// TIA Portal V18 export
DATA_BLOCK "SS1_A8_16DI_16DO_DI_Vars"   // DB11081
{ S7_Optimized_Access := 'FALSE' }
VERSION : 0.1
// stored: AutoNumber false, DBAccessibleFromOPCUA true, IsOnlyStoredInLoadMemory false, IsWriteProtectedInAS false
   VAR
      DI1 : "UDT_DIadv";
      DI2 : "UDT_DIadv";
      DI3 : "UDT_DIadv";
      DI4 : "UDT_DIadv";
      DI5 : "UDT_DIadv";
      DI6 : "UDT_DIadv";
      DI7 : "UDT_DIadv";
      DI8 : "UDT_DIadv";
      DI9 { S7_SetPoint := 'True'} : "UDT_DIadv";
      DI10 { S7_SetPoint := 'True'} : "UDT_DIadv";
      DI11 { S7_SetPoint := 'True'} : "UDT_DIadv";
      DI12 { S7_SetPoint := 'True'} : "UDT_DIadv";
      DI13 { S7_SetPoint := 'True'} : "UDT_DIadv";
      DI14 { S7_SetPoint := 'True'} : "UDT_DIadv";
      DI15 { S7_SetPoint := 'True'} : "UDT_DIadv";
      DI16 { S7_SetPoint := 'True'} : "UDT_DIadv";
   END_VAR
BEGIN
   DI1.cFuncSystemID := 1;
   DI1.cFuncVar := 11;
   DI2.cFuncSystemID := 1;
   DI3.cFuncSystemID := 1;
   DI4.cFuncSystemID := 1;
   DI4.cFuncVar := 6;
   DI5.cFuncSystemID := 1;
   DI5.cFuncVar := 4;
   DI6.cFuncSystemID := 1;
   DI6.cFuncVar := 21;
   DI7.cFuncSystemID := 1;
   DI8.cFuncSystemID := 1;
   DI9.cFuncSystemID := 1;
   DI10.cFuncSystemID := 3;
   DI10.cFuncVar := 13;
   DI11.cFuncSystemID := 3;
   DI12.cFuncSystemID := 3;
   DI13.cFuncSystemID := 3;
   DI13.cFuncVar := 3;
   DI14.cFuncSystemID := 3;
   DI14.cFuncVar := 3;
   DI15.cFuncSystemID := 3;
   DI15.cFuncVar := 14;
   DI16.cFuncSystemID := 3;
END_DATA_BLOCK
